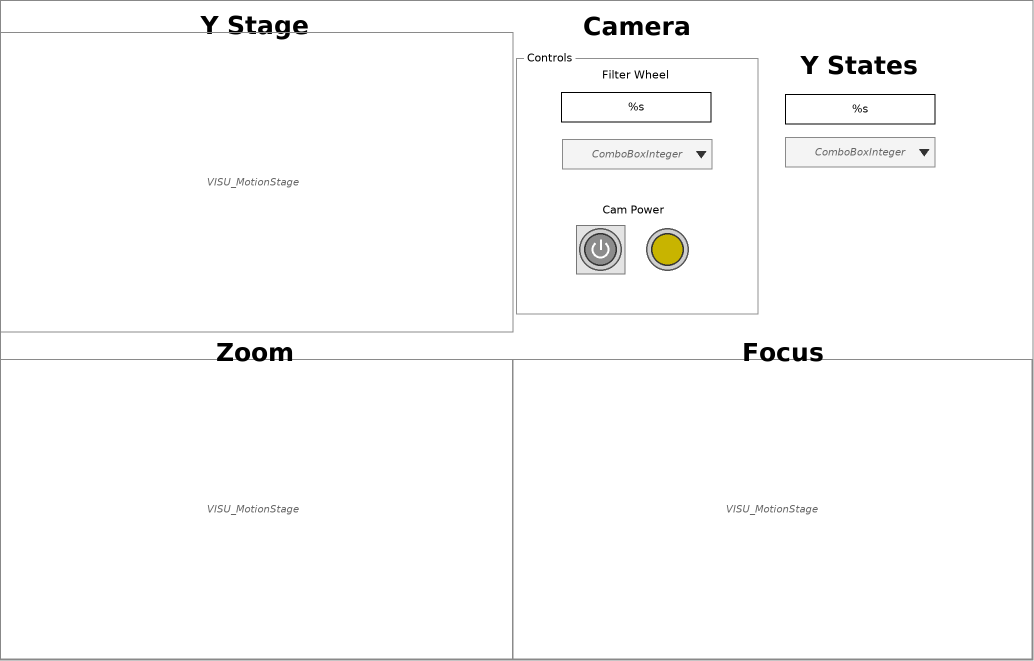
VISUALIZATION Visualization  // 1034x661
    Label (14,10 482x30), "Y Stage"
    Label (541,11 192x30), "Camera"
    GroupBox (516,50 242x264), "Controls"
        Lamp1 (127,175 49x49), variable: Main.fbXPIM.fbOpal.bOpalPowe, style: Lamp-Lamp1-Yellow
        PowerSwitch (60,175 49x49), variable: Main.fbXPIM.fbOpal.bOpalPower, behaviour: TOGGLE, style: Switch-PowerSwitch-Gray
        Label (39,145 157x30), "Cam Power"
        Rectangle (45,42 150x30), "%s", text variable: Main.fbXPIM.fbFilterWheel.nGetPos
        ComboBoxInteger (46,89 150x30), variable: Main.fbXPIM.fbFilterWheel.nSetPos, text list: 'TextListXPIMFilters'
        Label (41,10 157x30), "Filter Wheel"
    Frame (-7,32 520x300)
        shows VISU_MotionStage(VisuMotionStage := Main.M1, Extras := Main.M1_Extras)
    Frame (-7,359 520x300)
        shows VISU_MotionStage(VisuMotionStage := Main.M2, Extras := Main.M2_Extras)
    Frame (512,359 520x300)
        shows VISU_MotionStage(VisuMotionStage := Main.M3, Extras := Main.M3_Extras)
    Label (14,337 482x30), "Zoom"
    Label (542,337 482x30), "Focus"
    Label (787,50 145x30), "Y States"
    Rectangle (785,94 150x30), "%s", text variable: Main.fbXPIM.fbStates.enumGet
    ComboBoxInteger (785,137 150x30), variable: Main.fbXPIM.fbStates.enumSet, text list: 'TextListXPIMStates'
END_VISUALIZATION

(* stored: Version 1.1.0.1, ProductVersion 3.1.4022.18
   Visu Visualization: Id {af2f16f4-e7e7-4019-a84a-cc323e4115d2} *)
